INTERFACE I_Axis EXTENDS I_BaseAxis

PROPERTY isTracking : BOOL
GET
END_GET
END_PROPERTY

PROPERTY MoveAxis : BOOL
GET
END_GET
SET
END_SET
END_PROPERTY

PROPERTY MoveDone : BOOL
GET
END_GET
END_PROPERTY

PROPERTY SlewTime : LREAL
GET
END_GET
END_PROPERTY

PROPERTY StopAxis : BOOL
GET
END_GET
SET
END_SET
END_PROPERTY

PROPERTY Tracking : BOOL
GET
END_GET
SET
END_SET
END_PROPERTY

END_INTERFACE

(* stored: Version 1.1.0.1, ProductVersion 3.1.4024.15
   Itf I_Axis: Id {595a9217-864b-493b-b1f1-9dea5601aca8}
   Property isTracking: Id {0d2ea9c7-dd11-4be0-9e83-6118b37e161b}
   Get Get: Id {c9cdb742-ee96-4320-b6b2-cd6aece51d85}
   Property MoveAxis: Id {90f106f7-8dcd-4901-80fe-14c7f84618af}
   Get Get: Id {76723e17-1eb4-4ce1-b9ac-2b79b1a1f8b3}
   Set Set: Id {ca5e53e4-816b-479c-8ecd-bf8899ab3dee}
   Property MoveDone: Id {05c9ff68-0ac2-480d-ba33-0729891b3463}
   Get Get: Id {eaa34f86-7c88-4df7-aadc-db2e49929965}
   Property SlewTime: Id {ea9cbc59-52a8-43e3-b9ff-bd11e69913af}
   Get Get: Id {07820cdd-1819-4cf1-ad7a-493b97cc2472}
   Property StopAxis: Id {dda4b41f-dd83-495c-ad4d-1d299881860a}
   Get Get: Id {7a98b63c-6aab-43bf-a9c7-62fe5b2d1f52}
   Set Set: Id {0c3e415e-2ef7-4282-bb47-13c0b20ef9b1}
   Property Tracking: Id {79fcdc42-64ea-4f0e-bf51-0b2fee2f3261}
   Get Get: Id {adf4b757-aaba-4db1-8d0a-af3e137d0ff2}
   Set Set: Id {a7020af0-be07-460d-88fe-c9babbe577d5} *)
